{attribute 'GeneratedUsingTerminal: EL2521-0000-1019'}
{attribute addProperty BoxType "EL2521-0000-1019"}
{attribute addProperty Id "StatusAT %I*Status_5E172F147"}
{attribute addProperty CRC "1085474076"}
{attribute addProperty Size "7"}
TYPE PTO_Status_40B3051C :
STRUCT
	{attribute addProperty Name "Status"}
	Status AT %I* : Status_5E172F14;
END_STRUCT
END_TYPE

(* stored: Version 1.2.0.0, ProductVersion 3.1.4024.9
   DUT PTO_Status_40B3051C: Id {5f229d96-ee48-4fa7-83b3-1b1a8b4cce87} *)
